(* IEC 61131-3 sources: programs/VI-54/VI-54_20171205/VI-54_20171205/Stations/Screen/LseClass170718/Class/Management, 1 file *)

(* ---- Management.st ---- *)
(*!
<Class
	Name               = "Management"
	Revision           = "0.0"
	RealtimeTask       = "true"
	CyclicTask         = "false"
	BackgroundTask     = "false"
	Sigmatek           = "false"
	OSInterface        = "false"
	HighPriority       = "false"
	Automatic          = "false"
	UpdateMode         = "Prescan"
	SharedCommandTable = "true"
	Objectsize         = "(1080,120)">
	<Channels>
		<Server Name="__________" Visualized="false" Initialize="false" WriteProtected="true" Retentive="false"/>
		<Server Name="___________" Visualized="false" Initialize="false" WriteProtected="true" Retentive="false"/>
		<Server Name="AlarmActive" Visualized="true" Remotely="true" Initialize="false" WriteProtected="true" Retentive="false"/>
		<Server Name="ClassSvr" Visualized="false" Initialize="false" WriteProtected="true" Retentive="false"/>
		<Server Name="CleaningMode" Visualized="true" Initialize="false" WriteProtected="false" Retentive="false"/>
		<Server Name="Line_Runstatus" Visualized="true" Remotely="true" Initialize="false" WriteProtected="true" Retentive="false"/>
		<Server Name="Line_Speed" Visualized="true" Remotely="true" Initialize="false" WriteProtected="false" Retentive="false"/>
		<Server Name="Line_Started" Visualized="true" Initialize="false" WriteProtected="true" Retentive="false"/>
		<Server Name="Line_StartingUp" Visualized="false" Initialize="false" WriteProtected="true" Retentive="false"/>
		<Server Name="Line_Stopped" Visualized="true" Initialize="false" WriteProtected="true" Retentive="false"/>
		<Server Name="OverruleSafetyVI51" Visualized="true" Remotely="true" Initialize="true" WriteProtected="false" Retentive="File"/>
		<Server Name="ResetSignal" Visualized="true" Remotely="true" Initialize="false" WriteProtected="false" Retentive="false"/>
		<Client Name="Comm_Terminal" Required="true" Internal="false"/>
		<Client Name="iActRunStatus_VI49" Required="true" Internal="false"/>
		<Client Name="iActRunStatus_VI51" Required="true" Internal="false"/>
		<Client Name="iSafetyOK" Required="true" Internal="false"/>
		<Client Name="iStart" Required="true" Internal="false"/>
		<Client Name="iStop" Required="true" Internal="false"/>
		<Client Name="oResetAlarm" Required="true" Internal="false"/>
		<Client Name="Standard3" Required="true" Internal="true"/>
	</Channels>
	<Network Name="Management">
		<!-- List of Components in this network -->
		<Components>
			<Object
				Name           = "Standard3"
				Class          = "Standard"
				Position       = "(300,390)"
				Visualized     = "false"
				BackgroundTime = "1000 ms">
				<Channels>
					<Server Name="ClassSvr"/>
				</Channels>
			</Object>
		</Components>
		<Comments>
		</Comments>
		<!-- List of Connections in this network -->
		<Connections>
			<Connection Source="this.Standard3" Destination="Standard3.ClassSvr"/>
		</Connections>
		<!-- Headerfiles -->
		<Options>
		</Options>
	</Network>
</Class>
*)
Management : CLASS
  //Servers:
	ClassSvr 	: SvrChCmd_DINT;
	Line_Started 	: SvrCh_DINT;
	Line_Stopped 	: SvrCh_DINT;
	Line_StartingUp 	: SvrCh_DINT;
	CleaningMode 	: SvrCh_DINT;
	__________ 	: SvrCh_DINT;
	Line_Runstatus 	: SvrCh_RunningStateEnum;
	Line_Speed 	: SvrCh_DINT;
	ResetSignal 	: SvrCh_DINT;
	AlarmActive 	: SvrCh_DINT;
	___________ 	: SvrCh_DINT;
	OverruleSafetyVI51 	: SvrCh_DINT;
  //Clients:
	iSafetyOK 	: CltCh_DINT;
	iStart 	: CltCh_DINT;
	iStop 	: CltCh_DINT;
	Comm_Terminal 	: CltChCmd_TerminalControl;
	oResetAlarm 	: CltChCmd_AlarmDisplayList2;
	iActRunStatus_VI51 	: CltCh_RunningStateEnum;
	iActRunStatus_VI49 	: CltCh_RunningStateEnum;
	Standard3 	: CltChCmd_Standard;
  //Variables:
		LineRunstatusArray : ARRAY [0..cNbrOfMachinesInLine] OF RunningStateEnum;

		j 	: DINT;
		HoldReset 	: DINT;
		TmrHold 	: UDINT;
  //Functions:

	FUNCTION VIRTUAL GLOBAL RtWork
		VAR_INPUT
			EAX 	: UDINT;
		END_VAR
		VAR_OUTPUT
			state (EAX) 	: UDINT;
		END_VAR;

	FUNCTION GLOBAL CheckRunStatus
		VAR_INPUT
			InpStatus 	: RunningStateEnum;
		END_VAR
		VAR_OUTPUT
			OutputState 	: DINT;
		END_VAR;
  //Tables:
	FUNCTION @STD
		VAR_OUTPUT
			ret_code	: CONFSTATES;
		END_VAR;
	FUNCTION GLOBAL TAB @CT_;
END_CLASS;

#pragma using Standard
#pragma usingLtd AlarmDisplayList2
#pragma usingLtd TerminalControl

//

FUNCTION VIRTUAL GLOBAL Management::RtWork
	VAR_INPUT
		EAX 	: UDINT;
	END_VAR
	VAR_OUTPUT
		state (EAX) 	: UDINT;
	END_VAR

  // Read inputs & Runstatussen
  iSafetyOK          := iSafetyOK.Read();
  iStart             := iStart.Read();
  iStop              := iStop.Read();
  iActRunStatus_VI51 := iActRunStatus_VI51.Read();
  iActRunStatus_VI49 := iActRunStatus_VI49.Read();

  // Set all of the runstatussen in array
  LineRunstatusArray[1] := iActRunStatus_VI51;
  LineRunstatusArray[2] := iActRunStatus_VI49;

  // Check Safety Error
  AlarmActive := (Line_Runstatus = eNoodstopStatus | Line_Runstatus = eErrorStatus);

  // Set window start up
  if Standard3.R_TRIG(CLK:= Line_StartingUp) then
    Comm_Terminal.SelectWindowNbr(Nbr:= 105);
  elsif Standard3.F_TRIG(CLK:= Line_StartingUp) then
    Comm_Terminal.SelectWindow.Write(input:= -1);
  end_if;

  // Hold reset signal for at least 1000ms high
  if Standard3.TON(IN:= ResetSignal, PT:= 1000) then
    ResetSignal := 0;
  end_if;
  if ResetSignal = 1 then
    oResetAlarm.ResetData();
  end_if;
  if AlarmActive = 1 then // get alarm text
    oResetAlarm.HelpTxt.Write(input:= 0);
  end_if;

  // Runstatussen
  if CheckRunStatus(InpStatus:= eNoodstopStatus) = 1 then  // NOODSTOP
    Line_Started := 0;
    CleaningMode := 0;
    Line_StartingUp := 0;
    Line_Runstatus := eNoodstopStatus;
  elsif CheckRunStatus(InpStatus:= eErrorStatus) = 1 then // storing
    Line_Started := 0;
    CleaningMode := 0;
    Line_StartingUp := 0;
    Line_Runstatus := eErrorStatus;
  elsif iStop = 1 & (Line_Started = 1 | CleaningMode = 1) then // stop knop
    Line_Started := 0;
    CleaningMode := 0;
    Line_Runstatus := eStopStatus;
  elsif CleaningMode = 1 & Line_Started = 0 then  // machine in schoonmaak stand
    Line_Started := 0;
    Line_Runstatus := eCleaningStatus;
  elsif iStart = 1 & Line_Started = 0 then
    CleaningMode := 0;
    Line_Started := 1;
  else
    if Line_StartingUp = 1 then
      Line_Started := 0;
      if CheckRunStatus(InpStatus:= eStopStatus) = 1 then
        Line_StartingUp := 0;
      else
        Line_Runstatus := eStartUpStatus;
      end_if;
    elsif Line_Started = 1 then
      if CheckRunStatus(InpStatus:= eDriveOffStatus) = 1 then
        Line_Started := 0;  // na opstarten opnieuw start geven..
        Line_StartingUp := 1;
        Line_Runstatus := eStartUpStatus;
      else
        if Line_StartingUp = 0 then
          CleaningMode := 0;
          Line_Runstatus := eRunStatus;
        end_if;
      end_if;
    else
      Line_Runstatus := eStopStatus;
    end_if;
  end_if;
  Line_Stopped := (Line_Started = 0);

	state := READY;

END_FUNCTION

FUNCTION GLOBAL Management::CheckRunStatus
	VAR_INPUT
		InpStatus 	: RunningStateEnum;
	END_VAR
	VAR_OUTPUT
		OutputState 	: DINT;
	END_VAR
  VAR
  	i           : Dint;
  END_VAR

  OutputState := 0;
  j           := 0;

  Case InpStatus of
    eNoodstopStatus:
      for i := 1 to cNbrOfMachinesInLine do
        if LineRunstatusArray[i] = eNoodstopStatus then
          OutputState := 1;
        end_if;
      end_for;

    eErrorStatus:
      for i := 1 to cNbrOfMachinesInLine do
        if LineRunstatusArray[i] = eErrorStatus then
          OutputState := 1;
        end_if;
      end_for;

    eDriveOffStatus:
      for i := 1 to cNbrOfMachinesInLine do
        if LineRunstatusArray[i] = eDriveOffStatus then
          OutputState := 1;
        end_if;
      end_for;

    eStopStatus: // All of the belts are equeal to stopstatus
      for i := 1 to cNbrOfMachinesInLine do
        if LineRunstatusArray[i] = eStopStatus then
          j += 1;
          if j >= cNbrOfMachinesInLine then
            OutputState := 1;
          end_if;
        end_if;
      end_for;

  end_case;

END_FUNCTION
